Staubli VAL3: f1_cell_count.pgx

program f1_cell_count()
begin
  //given row,col , return position
  //retunr position
end
